// TwinCAT 3 PLC project TcCommando
// Title: TcCommando
// Company: Loupe
// Author: Loupe
// ProjectVersion: 0.0.5
// ProgramVersion: 3.1.4024.0
// libraries:
//   Tc2_Standard, * (Beckhoff Automation GmbH)
//   Tc2_System, * (Beckhoff Automation GmbH)
//   Tc3_Module, * (Beckhoff Automation GmbH)
//   TcPluginFramework, * (Loupe)
//   TcUnit, * (www.tcunit.org)
// project tree:
//   DUTs/ PLCopenCallGroupType.TcDUT, PLCopenCallInternal.TcDUT, PLCopenCallState.TcTLEO, PLCopenCommandInternal.TcDUT, PLCopenStatusBase.TcTLEO
//   GVLs/ GVLTcCommando.TcGVL
//   Interfaces/ IPLCopenBase.TcIO, IPLCopenCall.TcIO, IPLCopenCommand.TcIO, IPLCopenGroup.TcIO
//   / PlcTask.TcTTO
//   POUs/ PLCopenCall.TcPOU, PLCopenCallGroup.TcPOU, PLCopenCommand.TcPOU, PLCopenCommandGroup.TcPOU, PLCopenNullRemote.TcPOU
//   Test/ PLCopenCall_Test.TcPOU, TESTPRG.TcPOU, PLCopenCommand_Test.TcPOU
// real-time tasks:
//   TASK PlcTask: cycle T#10ms, priority 20, ADS port 350

CONFIGURATION TcCommando
    RESOURCE PLC ON TwinCAT3
        TASK PlcTask(INTERVAL := T#10ms, PRIORITY := 20);
        PROGRAM TESTPRG WITH PlcTask : TESTPRG;
    END_RESOURCE
END_CONFIGURATION

// ---- DUTs/PLCopenCallGroupType.TcDUT
TYPE
    PLCopenCallGroupType :
    STRUCT
        _startStep : ENUM; //The step when doStep was called
        _currentStep : ENUM;
        _lastRequestNumber : DINT;
        _onEntry : BOOL;
        _onExit : BOOL;
        _isDone : BOOL;
        _isAbort : BOOL;
        _isError : BOOL;
        _statusChecked : BOOL;
        _numberActiveCommands : INT;
        _commands : ARRAY[0..GVLTcCommando.MAX_RELATED_GROUPS] OF PLCopenCall;
        _syncAbort : BOOL;
        _syncError : BOOL;
        _syncDone : BOOL;
    END_STRUCT
END_TYPE

// ---- DUTs/PLCopenCallInternal.TcDUT
TYPE
    PLCopenCallInternal :
    STRUCT
        _state : PLCopenCallState;
        _Command : IPLCopenCommand;
        _abort : BOOL;
        _execute : BOOL;
        _break : BOOL;
        _RemoteStatus : PLCopenStatusBase;
        _self : IPLCopenCall;
    END_STRUCT
END_TYPE

// ---- DUTs/PLCopenCallState.TcTLEO
{attribute 'qualified_only'}
{attribute 'strict'}
TYPE PLCopenCallState :
(
	PLCOPEN_FUB_IDLE := 0,
	PLCOPEN_FUB_NEW_COMMAND,
	PLCOPEN_FUB_ABORTED,
	PLCOPEN_FUB_ABORT_OLD,
	PLCOPEN_FUB_STATUS,
	PLCOPEN_FUB_WRITE_PAR,
	PLCOPEN_FUB_SET_COMMAND,
	PLCOPEN_FUB_WORKING,
	PLCOPEN_FUB_CLEANUP,
	PLCOPEN_FUB_DONE
);
END_TYPE

// ---- DUTs/PLCopenCommandInternal.TcDUT
TYPE
    PLCopenCommandInternal :
    STRUCT
        _Execute : BOOL;
        _Trig : BOOL;
        _status : PLCopenStatusBase;
        _remote : IPLCopenCall;
        _nullRemote : PLCopenNullRemote;
        _commandGroups : ARRAY[0..GVLTcCommando.MAX_RELATED_GROUPS] OF IPLCopenGroup;
    END_STRUCT
END_TYPE

// ---- DUTs/PLCopenStatusBase.TcTLEO
{attribute 'qualified_only'}
TYPE PLCopenStatusBase :
(
	ERR_OK := 0,
	ERROR := 1,	
	ABORTED := 2,	
	ENABLED_WAITING := 65533,	
	NOT_ENABLED := 65534,	
	BUSY := 65535	
);
END_TYPE

// ---- GVLs/GVLTcCommando.TcGVL
{attribute 'qualified_only'}
VAR_GLOBAL
END_VAR
VAR_GLOBAL CONSTANT
    MAX_RELATED_GROUPS : USINT := 19;
END_VAR

// ---- Interfaces/IPLCopenBase.TcIO
// Copyright (c) 2024 Loupe (https://loupe.team), provided under the MIT License.

INTERFACE IPLCopenBase

PROPERTY Busy : BOOL
GET
END_GET
END_PROPERTY

PROPERTY ConsumeDone : Bool
GET
END_GET
END_PROPERTY

PROPERTY Done : BOOL
GET
END_GET
END_PROPERTY

PROPERTY Error : BOOL
GET
END_GET
END_PROPERTY

END_INTERFACE

// ---- Interfaces/IPLCopenCall.TcIO
// Copyright (c) 2024 Loupe (https://loupe.team), provided under the MIT License.

INTERFACE IPLCopenCall

METHOD Aborted : BOOL
VAR_INPUT
END_VAR
END_METHOD

METHOD Errored : BOOL
VAR_INPUT
    ID : INT;
END_VAR
END_METHOD

METHOD Finished : BOOL
VAR_INPUT
END_VAR
END_METHOD

METHOD Start : BOOL
VAR_INPUT
    Command : IPLCopenCommand;
END_VAR
END_METHOD

END_INTERFACE

// ---- Interfaces/IPLCopenCommand.TcIO
// Copyright (c) 2024 Loupe (https://loupe.team), provided under the MIT License.

INTERFACE IPLCopenCommand

METHOD Aborted : BOOL
VAR_INPUT
END_VAR
END_METHOD

METHOD AbortPreviousCommands : BOOL
VAR_INPUT
    newCommand : IPLCopenCommand;
END_VAR
END_METHOD

PROPERTY Consume : BOOL
GET
END_GET
END_PROPERTY

METHOD Errored : BOOL
VAR_INPUT
    ID : INT;
END_VAR
END_METHOD

PROPERTY Execute : BOOL
SET
END_SET
END_PROPERTY

METHOD Finished : BOOL
VAR_INPUT
END_VAR
END_METHOD

METHOD RegisterGroup : BOOL
VAR_INPUT
    group : IPLCopenGroup;
END_VAR
END_METHOD

{warning 'add property implementation'}
PROPERTY Remote : IPLCopenCall
GET
END_GET
SET
END_SET
END_PROPERTY

PROPERTY Status : PLCopenStatusBase
GET
END_GET
END_PROPERTY

END_INTERFACE

// ---- Interfaces/IPLCopenGroup.TcIO
// Copyright (c) 2024 Loupe (https://loupe.team), provided under the MIT License.

INTERFACE IPLCopenGroup

METHOD AbortPreviousCommands : BOOL
VAR_INPUT
    newCommand : IPLCopenCommand;
END_VAR
END_METHOD

END_INTERFACE

// ---- Test/TESTPRG.TcPOU
PROGRAM TESTPRG
VAR
    plcopenCommandTest : PLCopenCommand_Test;
    plcopenCallTest : PLCopenCall_Test;
END_VAR

// Copyright (c) 2024 Loupe (https://loupe.team), provided under the MIT License.

TcUnit.RUN();

END_PROGRAM

// ---- Test/PLCopenCommand_Test.TcPOU
FUNCTION_BLOCK PLCopenCommand_Test EXTENDS TcUnit.FB_TestSuite
VAR_INPUT
END_VAR
VAR_OUTPUT
END_VAR
VAR
END_VAR

// Copyright (c) 2024 Loupe (https://loupe.team), provided under the MIT License.

CallFinished();
CallAbort();
CallError();
AbortPrevious();

METHOD AbortPrevious
VAR
    command : PLCopenCommand();
    newCommand : PLCopenCommand();
END_VAR
// Copyright (c) 2024 Loupe (https://loupe.team), provided under the MIT License.

(*STweep.Disable*)

TEST('AbortPrevious');
	command.Execute := TRUE;
	command();
	command.AbortPreviousCommands(newCommand);
	
//	AssertEquals_INT(Expected := PLCopenStatusBase.ABORTED, Actual := command.status, Message := 'Initial command should be aborted');
TEST_FINISHED();
END_METHOD

METHOD CallAbort
VAR
    command : PLCopenCommand();
END_VAR
// Copyright (c) 2024 Loupe (https://loupe.team), provided under the MIT License.

(*STweep.Disable*)

TEST('CallAbort');
	AssertFalse(Condition := command.Consume, Message := 'Consume Should start false');
	AssertEquals_DINT(Actual := command.status, Expected:= PLCopenStatusBase.NOT_ENABLED, Message := 'Status should be not enabled');
	
	command.Execute := TRUE;
	
	AssertEquals_DINT(Actual := command.status, Expected:= PLCopenStatusBase.ENABLED_WAITING, Message := 'Status should be waiting');
	
	AssertTrue(Condition := command.Consume, Message := 'Consume Should start as true');
	AssertEquals_DINT(Actual := command.status, Expected:= PLCopenStatusBase.BUSY, Message := 'Status should be busy');
	
	AssertFalse(Condition := command.Consume, Message := 'Consume Should auto reset');
	AssertEquals_DINT(Actual := command.status, Expected:= PLCopenStatusBase.BUSY, Message := 'Status should be busy');
	
	command.Execute := TRUE;
	
	AssertEquals_DINT(Actual := command.status, Expected:= PLCopenStatusBase.ENABLED_WAITING, Message := 'Status should be waiting');
	
	AssertTrue(Condition := command.Consume, Message := 'Consume Should start as true after abort');
	AssertEquals_DINT(Actual := command.status, Expected:= PLCopenStatusBase.BUSY, Message := 'Status should be busy');
	
	AssertFalse(Condition := command.Consume, Message := 'Consume Should auto reset');
	AssertEquals_DINT(Actual := command.status, Expected:= PLCopenStatusBase.BUSY, Message := 'Status should be busy');
	
	command.Finished();
	
	AssertEquals_DINT(Actual := command.status, Expected:= PLCopenStatusBase.ERR_OK, Message := 'Status should be OK after finish');
	command();
	AssertEquals_DINT(Actual := command.status, Expected:= PLCopenStatusBase.NOT_ENABLED, Message := 'Status should auto reset');
	
	AssertFalse(Condition := command.Consume, Message := 'Consume Should auto reset');
	
TEST_FINISHED();
END_METHOD

METHOD CallError
VAR
    command : PLCopenCommand();
END_VAR
// Copyright (c) 2024 Loupe (https://loupe.team), provided under the MIT License.

(*STweep.Disable*)

TEST('CallError');

	AssertFalse(Condition := command.Consume, Message := 'Consume Should start false');
	AssertEquals_DINT(Actual := command.status, Expected:= PLCopenStatusBase.NOT_ENABLED, Message := 'Status should be not enabled');
	
	command.Execute := TRUE;
	
	AssertEquals_DINT(Actual := command.status, Expected:= PLCopenStatusBase.ENABLED_WAITING, Message := 'Status should be waiting');
	
	AssertTrue(Condition := command.Consume, Message := 'Consume Should start as true');
	AssertEquals_DINT(Actual := command.status, Expected:= PLCopenStatusBase.BUSY, Message := 'Status should be busy');
	
	AssertFalse(Condition := command.Consume, Message := 'Consume Should auto reset');
	AssertEquals_DINT(Actual := command.status, Expected:= PLCopenStatusBase.BUSY, Message := 'Status should be busy');
	
	command.Errored(PLCopenStatusBase.ERROR);
	
	AssertFalse(Condition := command.Consume, Message := 'Consume Should be false');
	AssertEquals_DINT(Actual := command.status, Expected:= PLCopenStatusBase.ERROR, Message := 'Status should be error');
	command();
	AssertEquals_DINT(Actual := command.status, Expected:= PLCopenStatusBase.NOT_ENABLED, Message := 'Status should auto reset');
	
	command.Finished();
	
	AssertEquals_DINT(Actual := command.status, Expected:= PLCopenStatusBase.NOT_ENABLED, Message := 'Status should be not enabled if it happens after error');
	
	AssertFalse(Condition := command.Consume, Message := 'Consume Should auto reset');

TEST_FINISHED();
END_METHOD

METHOD CallFinished
VAR
    command : PLCopenCommand();
END_VAR
// Copyright (c) 2024 Loupe (https://loupe.team), provided under the MIT License.

(*STweep.Disable*)

TEST('CallFinished');
	AssertFalse(Condition := command.Consume, Message := 'Consume should start false');
	AssertEquals_DINT(Actual := command.status, Expected:= PLCopenStatusBase.NOT_ENABLED, Message := 'Status should be not enabled');
	
	command.Execute := TRUE;
	
	AssertEquals_DINT(Actual := command.status, Expected:= PLCopenStatusBase.ENABLED_WAITING, Message := 'Status should be waiting');
	
	AssertTrue(Condition := command.Consume, Message := 'Consume should start as true');
	AssertEquals_DINT(Actual := command.status, Expected:= PLCopenStatusBase.BUSY, Message := 'Status should be busy');
	
	AssertFalse(Condition := command.Consume, Message := 'Consume should auto reset');
	AssertEquals_DINT(Actual := command.status, Expected:= PLCopenStatusBase.BUSY, Message := 'Status should be busy');
	
	command.Finished();
	AssertEquals_DINT(Actual := command.status, Expected:= PLCopenStatusBase.ERR_OK, Message := 'Status should be OK after finish');
	command();
	AssertEquals_DINT(Actual := command.status, Expected:= PLCopenStatusBase.NOT_ENABLED, Message := 'Status should auto reset');
	
	AssertFalse(Condition := command.Consume, Message := 'Consume should auto reset');

TEST_FINISHED();
END_METHOD

END_FUNCTION_BLOCK

// ---- POUs/PLCopenCommand.TcPOU
FUNCTION_BLOCK PLCopenCommand IMPLEMENTS IPLCopenCommand
VAR
    _PLCopenCommand : PLCopenCommandInternal;
END_VAR

// Copyright (c) 2024 Loupe (https://loupe.team), provided under the MIT License.

IF _PLCopenCommand._status <> PLCopenStatusBase.BUSY AND NOT Execute THEN
    _PLCopenCommand._status := PLCopenStatusBase.NOT_ENABLED;
END_IF

METHOD Aborted : BOOL
VAR_INPUT
END_VAR
// Copyright (c) 2024 Loupe (https://loupe.team), provided under the MIT License.

_PLCopenCommand._status := PLCopenStatusBase.ABORTED;

Remote.Aborted();
Remote := 0;
END_METHOD

METHOD AbortPreviousCommands : BOOL
VAR_INPUT
    newCommand : IPLCopenCommand;
END_VAR
VAR
    i : USINT;
END_VAR
// Copyright (c) 2024 Loupe (https://loupe.team), provided under the MIT License.

//If there is a remote, abort it here
//Don't use this^.abort() because we don't want about ourselves
Remote.Aborted();
Remote := 0;

//Abort any related commands
FOR i := 0 TO GVLTcCommando.MAX_RELATED_GROUPS DO
    IF _PLCopenCommand._commandGroups[i] <> 0 THEN
        _PLCopenCommand._commandGroups[i].AbortPreviousCommands(newCommand);
    END_IF
END_FOR
END_METHOD

METHOD FINAL BaseSize : ULINT
// Copyright (c) 2024 Loupe (https://loupe.team), provided under the MIT License.

BaseSize := SIZEOF(THIS^);
END_METHOD

PROPERTY Consume : BOOL
GET
// Copyright (c) 2024 Loupe (https://loupe.team), provided under the MIT License.

Consume := _PLCopenCommand._Execute;

IF _PLCopenCommand._Execute THEN
    //	THIS^.AbortPreviousCommands( THIS^ );//This is meant to abort if the command comes locally
    _PLCopenCommand._status := PLCopenStatusBase.BUSY;
END_IF

_PLCopenCommand._Execute := FALSE;
END_GET
END_PROPERTY

METHOD Errored : BOOL
VAR_INPUT
    ID : INT;
END_VAR
// Copyright (c) 2024 Loupe (https://loupe.team), provided under the MIT License.

CASE ID OF
    //Any of these statuses are invalid to return as an error.
    //Override to error
    PLCopenStatusBase.BUSY,
        PLCopenStatusBase.ENABLED_WAITING,
        PLCopenStatusBase.ERR_OK:
        _PLCopenCommand._status := PLCopenStatusBase.ERROR;
ELSE
    //Any other status can be passed through
    _PLCopenCommand._status := ID;
END_CASE

Remote.Errored(ID);
END_METHOD

{attribute 'monitoring' := 'call'}
PROPERTY Execute : BOOL
GET
// Copyright (c) 2024 Loupe (https://loupe.team), provided under the MIT License.

Execute := _PLCopenCommand._Execute;
END_GET
SET
// Copyright (c) 2024 Loupe (https://loupe.team), provided under the MIT License.

//We are already executing
IF _PLCopenCommand._Trig = TRUE AND Execute = TRUE THEN

    ; //Do nothing
    //Trigger an execute
ELSIF _PLCopenCommand._Trig = FALSE AND Execute = TRUE THEN
    _PLCopenCommand._status := PLCopenStatusBase.ENABLED_WAITING;
    _PLCopenCommand._Execute := TRUE;

    THIS^.AbortPreviousCommands(THIS^); //This is meant to abort if the command comes locally	

    // We were executing, but resetting it to false;
    // Just resetting execute to false all the time is OK
ELSIF Execute = FALSE THEN
    _PLCopenCommand._Execute := FALSE;
END_IF
END_SET
END_PROPERTY

METHOD FB_init : BOOL
VAR_INPUT
    bInitRetains : BOOL; // if TRUE, the retain variables are initialized (warm start / cold start)
    bInCopyCode : BOOL; // if TRUE, the instance afterwards gets moved into the copy code (online change)
END_VAR
// Copyright (c) 2024 Loupe (https://loupe.team), provided under the MIT License.

_PLCopenCommand._status := PLCopenStatusBase.NOT_ENABLED;
END_METHOD

METHOD Finished : BOOL
VAR_INST
    derived : BOOL;
END_VAR
// Copyright (c) 2024 Loupe (https://loupe.team), provided under the MIT License.

IF _PLCopenCommand._status = PLCopenStatusBase.BUSY THEN
    _PLCopenCommand._status := PLCopenStatusBase.ERR_OK;
END_IF

Remote.Finished();
END_METHOD


METHOD GetSize : ULINT
// Copyright (c) 2024 Loupe (https://loupe.team), provided under the MIT License.

GetSize := SIZEOF(THIS^);
END_METHOD

METHOD GetThis : ULINT
// Copyright (c) 2024 Loupe (https://loupe.team), provided under the MIT License.

GetThis := THIS;
END_METHOD

METHOD RegisterGroup : BOOL
VAR_INPUT
    group : IPLCopenGroup;
END_VAR

VAR
    i : INT;
END_VAR
// Copyright (c) 2024 Loupe (https://loupe.team), provided under the MIT License.

FOR i := 0 TO GVLTcCommando.MAX_RELATED_GROUPS DO
    IF _PLCopenCommand._commandGroups[i] = 0 THEN
        _PLCopenCommand._commandGroups[i] := group;
        EXIT;
    END_IF
END_FOR
END_METHOD

PROPERTY Remote : IPLCopenCall
GET
// Copyright (c) 2024 Loupe (https://loupe.team), provided under the MIT License.

IF _PLCopenCommand._remote <> 0 THEN
    Remote := _PLCopenCommand._remote;
ELSE
    Remote := _PLCopenCommand._nullRemote;
END_IF
END_GET
SET
// Copyright (c) 2024 Loupe (https://loupe.team), provided under the MIT License.

_PLCopenCommand._remote := Remote;
END_SET
END_PROPERTY

{attribute 'monitoring' := 'call'}
PROPERTY Status : PLCopenStatusBase
GET
// Copyright (c) 2024 Loupe (https://loupe.team), provided under the MIT License.

status := _PLCopenCommand._status;
END_GET
END_PROPERTY

END_FUNCTION_BLOCK

// ---- Test/PLCopenCall_Test.TcPOU
FUNCTION_BLOCK PLCopenCall_Test EXTENDS FB_TestSuite
VAR_INPUT
END_VAR
VAR_OUTPUT
END_VAR
VAR
END_VAR

// Copyright (c) 2024 Loupe (https://loupe.team), provided under the MIT License.

Abort();
Call();
Clear();
Exec();
Start();

METHOD Abort
VAR
    call1 : PLCopenCall();
    call2 : PLCopenCall();
    command : PLCopenCommand();
END_VAR
// Copyright (c) 2024 Loupe (https://loupe.team), provided under the MIT License.

(*STweep.Disable*)

TEST('Abort');
	
	call1();
	call2();

	call1.Exec(command);
	call1.Execute := FALSE;

	AssertEquals_INT(call1.Status, PLCopenStatusBase.BUSY, Message := 'Status should be busy');
	AssertEquals_INT(call2.Status, PLCopenStatusBase.NOT_ENABLED, Message := 'Status should be not enabled');

	AssertTrue(command.Execute, Message := 'Execute should be true on command');
	AssertEquals_INT(command.Status, PLCopenStatusBase.ENABLED_WAITING, Message := 'First command should be waiting');
	
	AssertTrue(command.Consume, Message := 'consume should be true');
	AssertFalse(command.Consume, Message := 'consume should be false on second read');
	AssertEquals_INT(command.Status, PLCopenStatusBase.BUSY, Message := 'Command should be busy');

	call2.Exec(Command);
	call2.Execute := FALSE;

	call1();
	AssertEquals_INT(call1.Status, PLCopenStatusBase.ABORTED, Message := 'Status should be aborted');
	AssertEquals_INT(call2.Status, PLCopenStatusBase.BUSY, Message := 'Status should be busy');

	AssertTrue(command.Execute, Message := 'Execute should be true on command');
	AssertEquals_INT(command.Status, PLCopenStatusBase.ENABLED_WAITING, Message := 'First command should be waiting');
	
	AssertTrue(command.Consume, Message := 'consume should be true');
	AssertFalse(command.Consume, Message := 'consume should be false on second read');
	AssertEquals_INT(command.Status, PLCopenStatusBase.BUSY, Message := 'Command should be busy');

	command.Finished();
	
	call1();
	call2();

	AssertEquals_INT(call1.Status, PLCopenStatusBase.NOT_ENABLED, Message := 'Status should be no enabled');
	AssertEquals_INT(call2.Status, PLCopenStatusBase.ERR_OK, Message := 'Status should be err ok');
	
	

TEST_FINISHED();
END_METHOD

METHOD Call
VAR
    call : PLCopenCall;
    command : PLCopenCommand;
END_VAR
// Copyright (c) 2024 Loupe (https://loupe.team), provided under the MIT License.

(*STweep.Disable*)

TEST('PLCopenCallIdle');

	AssertFalse(Condition := call.Busy, Message := 'Busy should be false as default');
	AssertFalse(Condition := call.Done, Message := 'Done should be false as default');
	AssertFalse(Condition := call.Error, Message := 'Error should be false as default');
	
	call.Exec(command);
	AssertTrue(Condition := call.Busy, Message := 'Busy should be true after first exec');
	AssertFalse(Condition := call.Done, Message := 'Done should be false after first exec');
	AssertFalse(Condition := call.Error, Message := 'Error should be false as default');
	AssertEquals_DINT(Expected := PLCopenStatusBase.BUSY, Actual := call.Status, Message := 'Status should be FUB Working');

// new command

// this command aborted

// cleanup

// done

// working

// aborted

// TODO multiple calls
TEST_FINISHED();
END_METHOD

METHOD Clear
VAR
    call : PLCopenCall();
    status : PLCopenStatusBase;
END_VAR
// Copyright (c) 2024 Loupe (https://loupe.team), provided under the MIT License.

(*STweep.Disable*)

TEST('Clear');
	call.Execute := TRUE;
	call();
	status := call.Clear();
	AssertFalse(call.Execute, Message := 'Execute should not be true');
	AssertEquals_INT(Expected := PLCopenStatusBase.NOT_ENABLED, Actual := status, Message := 'Call status should be not enabled');
TEST_FINISHED();
END_METHOD

METHOD Errored
VAR_INPUT
END_VAR
// Copyright (c) 2024 Loupe (https://loupe.team), provided under the MIT License.

(*STweep.Disable*)
END_METHOD

METHOD Exec
VAR
    call : PLCopenCall();
    command1 : PLCopenCommand();
    command2 : PLCopenCommand();
END_VAR
// Copyright (c) 2024 Loupe (https://loupe.team), provided under the MIT License.

(*STweep.Disable*)

TEST('Exec1');

	call.Exec(command1);
	AssertTrue(call.Execute, Message := 'Execute should be true on call');
	AssertTrue(command1.Execute, Message := 'Execute should be true on command');
	AssertEquals_INT(command1.Status, PLCopenStatusBase.ENABLED_WAITING, Message := 'First command should be aborted');
	AssertEquals_INT(command2.Status, PLCopenStatusBase.NOT_ENABLED, Message := 'Second command should be not enabled');
	
	AssertTrue(command1.Consume, Message := 'First command consume should be true');
	AssertFalse(command2.Consume, Message := 'Second command consume should be false');

	AssertFalse(command1.Consume, Message := 'First command consume should be false');
	AssertFalse(command2.Consume, Message := 'Second command consume should be false');

	command1.Finished();

	call();

	AssertEquals_INT(call.Status, PLCopenStatusBase.ERR_OK, Message := 'Call should be Err OK');
	AssertEquals_INT(command1.Status, PLCopenStatusBase.ERR_OK, Message := 'First command should be Err OK');
	AssertEquals_INT(command2.Status, PLCopenStatusBase.NOT_ENABLED, Message := 'Second command should be enabled waiting');
TEST_FINISHED();
TEST('Exec2');
	
//	call.Clear();//DO we need clear?


	call.Exec(command2);

//	AssertEquals_INT(command1.Status, PLCopenStatusBase.NOT_ENABLED, Message := 'First command should be Not Enabled');//This is actually not defined, the status doesn't get reset until it's needed again
	AssertEquals_INT(command2.Status, PLCopenStatusBase.ENABLED_WAITING, Message := 'Second command should be enabled waiting');

	AssertFalse(command1.Consume, Message := 'First command consume should be false');
	AssertTrue(command2.Consume, Message := 'Second command consume should be true');

	AssertFalse(command1.Consume, Message := 'First command consume should be false');
	AssertFalse(command2.Consume, Message := 'Second command consume should be false');

	command2.Finished();

	call();

	AssertEquals_INT(call.Status, PLCopenStatusBase.ERR_OK, Message := 'Call should be Err OK');
//	AssertEquals_INT(command1.Status, PLCopenStatusBase.NOT_ENABLED, Message := 'First command should be Not Enabled');//This is actually not defined, the status doesn't get reset until it's needed again
	AssertEquals_INT(command2.Status, PLCopenStatusBase.ERR_OK, Message := 'Second command should be ERR OK');

	
	call.Exec(command1);
	AssertEquals_INT(command1.Status, PLCopenStatusBase.ENABLED_WAITING, Message := 'First command should be enabled waiting');
//	AssertEquals_INT(command2.Status, PLCopenStatusBase.NOT_ENABLED, Message := 'Second command should be not enabled');//This is actually not defined, the status doesn't get reset until it's needed again

TEST_FINISHED();
END_METHOD

METHOD Start
VAR
    call : PLCopenCall();
    command1 : PLCopenCommand();
    command2 : PLCopenCommand();
END_VAR
// Copyright (c) 2024 Loupe (https://loupe.team), provided under the MIT License.

(*STweep.Disable*)

TEST('Start');

	call.Start(command1);
	AssertTrue(command1.Execute, Message := 'Execute should be true');
	
	call.Start(command2);
	AssertTrue(command2.Execute, Message := 'Execute should be true');

TEST_FINISHED();
END_METHOD

END_FUNCTION_BLOCK

// ---- POUs/PLCopenCall.TcPOU
FUNCTION_BLOCK PLCopenCall IMPLEMENTS IPLCopenCall
VAR_INPUT
    Execute : BOOL;
    Command : IPLCopenCommand;
    Fallback : PLCopenStatusBase;
END_VAR
VAR_OUTPUT
    Status : PLCopenStatusBase;
    Busy : BOOL;
    Done : BOOL;
    Error : BOOL;
    CommandAborted : BOOL;
END_VAR
VAR
    _PLCopenCallInternal : PLCopenCallInternal;
END_VAR

// Copyright (c) 2024 Loupe (https://loupe.team), provided under the MIT License.

Call();

METHOD Aborted : BOOL
// Copyright (c) 2024 Loupe (https://loupe.team), provided under the MIT License.

_PLCopenCallInternal._abort := true;
END_METHOD

METHOD Call : BOOL
VAR
    _break : BOOL;
END_VAR
// Copyright (c) 2024 Loupe (https://loupe.team), provided under the MIT License.

//Capture edges
IF NOT Execute THEN
    _PLCopenCallInternal._execute := FALSE;
END_IF

// Start a new command on edge
IF (Execute AND NOT _PLCopenCallInternal._execute) THEN
    _PLCopenCallInternal._execute := TRUE;
    _PLCopenCallInternal._state := PLCopenCallState.PLCOPEN_FUB_NEW_COMMAND;
END_IF

// If this call get aborted, handle it
IF (_PLCopenCallInternal._abort) THEN
    _PLCopenCallInternal._abort := 0;
    _PLCopenCallInternal._state := PLCopenCallState.PLCOPEN_FUB_ABORTED;
END_IF

_PLCopenCallInternal._self := THIS^;

// Use a "while not break" to enable multiple passes on the state machine,
// to do as much as possible in a single call	
_break := FALSE;

WHILE _break = FALSE DO
    CASE (_PLCopenCallInternal._state) OF

        // IDLE
        PLCopenCallState.PLCOPEN_FUB_IDLE:
            Status := PLCopenStatusBase.NOT_ENABLED;
            Busy := FALSE;
            Done := FALSE;
            Error := FALSE;
            CommandAborted := FALSE;
            _break := TRUE;

        // Start a new command
        PLCopenCallState.PLCOPEN_FUB_NEW_COMMAND:
            Status := PLCopenStatusBase.BUSY;
            _PLCopenCallInternal._RemoteStatus := PLCopenStatusBase.BUSY;
            Busy := TRUE;
            Done := FALSE;
            Error := FALSE;
            CommandAborted := FALSE;

            // If this call is the current command:
            // 1. don't need feedback (TODO why? because it is being aborted?)
            // 2. this call doesn't get the abort
            // so remove this FUB before calling abort previous
            IF _PLCopenCallInternal._Command <> 0 THEN
                IF _PLCopenCallInternal._Command.Remote = _PLCopenCallInternal._self THEN
                    _PLCopenCallInternal._Command.Remote := 0;
                END_IF
            END_IF

            // Get the new command
            _PLCopenCallInternal._command := Command;

            IF _PLCopenCallInternal._Command <> 0 THEN
                _PLCopenCallInternal._state := PLCopenCallState.PLCOPEN_FUB_ABORT_OLD;
                // No _break
            ELSE
                _PLCopenCallInternal._state := PLCopenCallState.PLCOPEN_FUB_WORKING;
                _PLCopenCallInternal._RemoteStatus := Fallback;
                _break := TRUE;
            END_IF
        // No _break

        // Abort any commands that were active using the same PLCopen state
        PLCopenCallState.PLCOPEN_FUB_ABORT_OLD:
            _PLCopenCallInternal._Command.AbortPreviousCommands(_PLCopenCallInternal._Command);

            _PLCopenCallInternal._state := PLCopenCallState.PLCOPEN_FUB_SET_COMMAND;
        //no break;

        // Start the command
        PLCopenCallState.PLCOPEN_FUB_SET_COMMAND:
            _PLCopenCallInternal._Command.Execute := TRUE;
            _PLCopenCallInternal._Command.Remote := THIS^;

            Busy := TRUE;
            _PLCopenCallInternal._state := PLCOpenCallState.PLCOPEN_FUB_WORKING;
        // No _break

        //Wait for the command to be finished
        PLCopenCallState.PLCOPEN_FUB_WORKING:
            Busy := TRUE;
            // No _break

            IF (_PLCopenCallInternal._RemoteStatus <> PLCopenStatusBase.BUSY AND
                _PLCopenCallInternal._RemoteStatus <> PLCopenStatusBase.ENABLED_WAITING) THEN
                Status := _PLCopenCallInternal._RemoteStatus;
                Busy := FALSE;

                IF (Status = 0) THEN
                    Done := TRUE;

                ELSE
                    Error := TRUE;
                END_IF

                _PLCopenCallInternal._state := PLCopenCallState.PLCOPEN_FUB_CLEANUP;
                // No _break
            ELSE
                _break := TRUE;
            END_IF

        PLCopenCallState.PLCOPEN_FUB_CLEANUP:
            // Remove self from the source command
            IF _PLCopenCallInternal._Command <> 0 THEN
                _PLCopenCallInternal._Command.Remote := 0;
                _PLCopenCallInternal._Command := 0;
            END_IF

            _PLCopenCallInternal._state := PLCopenCallState.PLCOPEN_FUB_DONE;
            // Break to force at least 1 cycle with statuses
            _break := TRUE;

        PLCopenCallState.PLCOPEN_FUB_DONE:

            IF (NOT Execute) THEN
                _PLCopenCallInternal._state := PLCopenCallState.PLCOPEN_FUB_IDLE;
                Status := PLCopenStatusBase.NOT_ENABLED;
                Busy := FALSE;
                Done := FALSE;
                Error := FALSE;
                CommandAborted := FALSE;
            END_IF

            _break := TRUE;

        PLCopenCallState.PLCOPEN_FUB_ABORTED:
            Status := PLCopenStatusBase.ABORTED;
            Busy := FALSE;
            Done := FALSE;
            Error := FALSE;
            CommandAborted := TRUE;
            _PLCopenCallInternal._command := 0;
            _PLCopenCallInternal._state := PLCopenCallState.PLCOPEN_FUB_DONE;
            _break := TRUE;

    END_CASE
END_WHILE
END_METHOD

METHOD Clear : PLCopenStatusBase
// Copyright (c) 2024 Loupe (https://loupe.team), provided under the MIT License.

THIS^.Execute := FALSE;
THIS^._PLCopenCallInternal._state := PLCopenCallState.PLCOPEN_FUB_CLEANUP;
//One call to cleanup
THIS^.Call();
//Second call to clear
THIS^.Call();
Clear := THIS^.Status;
END_METHOD

METHOD Errored : BOOL
VAR_INPUT
    ID : INT;
END_VAR
// Copyright (c) 2024 Loupe (https://loupe.team), provided under the MIT License.

CASE ID OF
    //Any of these statuses are invalid to return as an error.
    //Override to error
    PLCopenStatusBase.BUSY,
        PLCopenStatusBase.ENABLED_WAITING,
        PLCopenStatusBase.ERR_OK:
        _PLCopenCallInternal._RemoteStatus := PLCopenStatusBase.ERROR;
ELSE
    //Any other status can be passed through
    _PLCopenCallInternal._RemoteStatus := ID;
END_CASE
END_METHOD

METHOD Exec : PLCopenStatusBase
VAR_INPUT
    Command : IPLCopenCommand;
END_VAR
// Copyright (c) 2024 Loupe (https://loupe.team), provided under the MIT License.

//Call with false to force an edge
//	This will also Abort the previous command if it exists
THIS^.Execute := FALSE;
THIS^.Call();

THIS^.Command := Command;
THIS^.Execute := TRUE;
THIS^.Call();
Exec := THIS^.Status;
END_METHOD

METHOD Finished : BOOL
// Copyright (c) 2024 Loupe (https://loupe.team), provided under the MIT License.

_PLCopenCallInternal._RemoteStatus := PLCopenStatusBase.ERR_OK;
END_METHOD

METHOD Start : BOOL
VAR_INPUT
    Command : IPLCopenCommand;
END_VAR
// Copyright (c) 2024 Loupe (https://loupe.team), provided under the MIT License.

THIS^.Exec(Command);
END_METHOD

END_FUNCTION_BLOCK

// ---- POUs/PLCopenCallGroup.TcPOU
FUNCTION_BLOCK PLCopenCallGroup IMPLEMENTS IPLCopenCall
VAR_INPUT
END_VAR
VAR_OUTPUT
END_VAR
VAR
    _callGroup : PLCopenCallGroupType;
END_VAR

// Copyright (c) 2024 Loupe (https://loupe.team), provided under the MIT License.

METHOD Aborted : BOOL
// Copyright (c) 2024 Loupe (https://loupe.team), provided under the MIT License.

_callGroup._syncAbort := TRUE;
END_METHOD

METHOD PRIVATE CheckStatus : BOOL
VAR
    _commandIndex : INT;
    _anyAbort : BOOL;
    _anyBusy : BOOL;
    _anyError : BOOL;
END_VAR
// Copyright (c) 2024 Loupe (https://loupe.team), provided under the MIT License.

//If it's not in the list
FOR _commandIndex := 0 TO GVLTcCommando.MAX_RELATED_GROUPS DO
    IF _callGroup._commands[_commandIndex].Command <> 0 THEN
        _callGroup._commands[_commandIndex]();

        IF _callGroup._commands[_commandIndex].CommandAborted THEN
            _anyAbort := TRUE;
        ELSIF _callGroup._commands[_commandIndex].Error THEN
            _anyError := TRUE;
        ELSIF _callGroup._commands[_commandIndex].Busy THEN
            _anyBusy := TRUE;
        ELSE
            _callGroup._commands[_commandIndex].Command := 0;
        END_IF
    END_IF
END_FOR

_callGroup._isError := FALSE;
_callGroup._isAbort := FALSE;
_callGroup._isDone := FALSE;

IF _anyError OR _callGroup._syncError THEN
    _callGroup._isError := TRUE;
ELSIF _anyAbort OR _callGroup._syncAbort THEN
    _callGroup._isAbort := TRUE;
ELSIF NOT _anyBusy THEN
    _callGroup._isDone := TRUE;
END_IF
END_METHOD

METHOD Errored : BOOL
VAR_INPUT
    ID : INT;
END_VAR
// Copyright (c) 2024 Loupe (https://loupe.team), provided under the MIT License.

_callGroup._syncError := TRUE;
END_METHOD

METHOD Finished : BOOL
// Copyright (c) 2024 Loupe (https://loupe.team), provided under the MIT License.

_callGroup._syncDone := TRUE;
END_METHOD

PROPERTY IsAbort : BOOL
GET
// Copyright (c) 2024 Loupe (https://loupe.team), provided under the MIT License.

CheckStatus();
IsAbort := _callGroup._isAbort;
END_GET
END_PROPERTY

PROPERTY IsDone : BOOL
GET
// Copyright (c) 2024 Loupe (https://loupe.team), provided under the MIT License.

CheckStatus();

//Check if we are done
IsDone := _callGroup._isDone;
END_GET
END_PROPERTY

PROPERTY IsError : BOOL
GET
// Copyright (c) 2024 Loupe (https://loupe.team), provided under the MIT License.

CheckStatus();

IsError := _callGroup._isError;
END_GET
END_PROPERTY

{warning 'add method implementation '}
METHOD PLCopenCall : PLCopenStatusBase
VAR_INPUT
    Command : IPLCopenCommand;
END_VAR
// Copyright (c) 2024 Loupe (https://loupe.team), provided under the MIT License.
END_METHOD

METHOD ResetCommands : BOOL
VAR
    _commandIndex : INT;
END_VAR
// Copyright (c) 2024 Loupe (https://loupe.team), provided under the MIT License.

//If it's not in the list
FOR _commandIndex := 0 TO GVLTcCommando.MAX_RELATED_GROUPS DO
    _callGroup._commands[_commandIndex].Clear();
END_FOR
END_METHOD

METHOD Start : BOOL
VAR_INPUT
    Command : IPLCopenCommand;
END_VAR
VAR
    _commandIndex : INT;
END_VAR
// Copyright (c) 2024 Loupe (https://loupe.team), provided under the MIT License.

// Check if it's already in the list
FOR _commandIndex := 0 TO GVLTcCommando.MAX_RELATED_GROUPS DO
    IF _callGroup._commands[_commandIndex].Command = Command THEN
        _callGroup._commands[_commandIndex].Exec(Command);
        Start := TRUE;
        RETURN;
    END_IF
END_FOR

// If it's not in the list
FOR _commandIndex := 0 TO GVLTcCommando.MAX_RELATED_GROUPS DO
    IF _callGroup._commands[_commandIndex].Command = 0 THEN
        _callGroup._commands[_commandIndex].Exec(Command);
        Start := TRUE;
        RETURN;
    END_IF
END_FOR

Start := FALSE;

//TODO: All out of commands.. Throw an error
END_METHOD

END_FUNCTION_BLOCK

// ---- POUs/PLCopenCommandGroup.TcPOU
{attribute 'call_after_init'}
FUNCTION_BLOCK PLCopenCommandGroup IMPLEMENTS IPLCopenGroup
VAR_INPUT
    commands : ARRAY[0..GVLTcCommando.MAX_RELATED_GROUPS] OF IPLCopenCommand;
END_VAR

// Copyright (c) 2024 Loupe (https://loupe.team), provided under the MIT License.

METHOD AbortPreviousCommands : BOOL
VAR_INPUT
    newCommand : IPLCopenCommand;
END_VAR

VAR
    i : INT;
END_VAR
// Copyright (c) 2024 Loupe (https://loupe.team), provided under the MIT License.

FOR i := 0 TO GVLTcCommando.MAX_RELATED_GROUPS DO

    IF commands[i] <> 0 AND commands[i] <> newCommand THEN

        commands[i].Aborted();

    END_IF

END_FOR
END_METHOD

{attribute 'call_after_init'}
METHOD RegisterCommands : BOOL
VAR
    i : INT;
END_VAR
// Copyright (c) 2024 Loupe (https://loupe.team), provided under the MIT License.

ADSLOGSTR(msgCtrlMask := ADSLOG_MSGTYPE_ERROR,
    msgFmtStr := 'Initing command group',
    strArg := '');

FOR i := 0 TO GVLTcCommando.MAX_RELATED_GROUPS DO

    IF commands[i] <> 0 THEN

        commands[i].registerGroup(THIS^);

    END_IF

END_FOR
END_METHOD

END_FUNCTION_BLOCK

// ---- POUs/PLCopenNullRemote.TcPOU
FUNCTION_BLOCK PLCopenNullRemote IMPLEMENTS IPLCopenCall

// Copyright (c) 2024 Loupe (https://loupe.team), provided under the MIT License.

METHOD Aborted : BOOL
// Copyright (c) 2024 Loupe (https://loupe.team), provided under the MIT License.
END_METHOD

METHOD Errored : BOOL
VAR_INPUT
    ID : INT;
END_VAR
// Copyright (c) 2024 Loupe (https://loupe.team), provided under the MIT License.
END_METHOD

METHOD Finished : BOOL
// Copyright (c) 2024 Loupe (https://loupe.team), provided under the MIT License.
END_METHOD

{warning 'add method implementation '}
METHOD Start : BOOL
VAR_INPUT
    Command : IPLCopenCommand;
END_VAR
// Copyright (c) 2024 Loupe (https://loupe.team), provided under the MIT License.

//TODO
END_METHOD

END_FUNCTION_BLOCK
